TYPE (* IEC61131-3, Table 14#5 *)
  (* Standard: 1131-3 *)
  (* Version 0.0, 1/8/2024, Cheyan, Schneider Electric, Template *)
  PACKAGE Main;
  {SET_ATTRIBUTE(nxtDataType, QdpEwqSPB7qzzh+NTQEinmNZ98ZHkHWxvNuG/cIXeimh6FQ57YZhv3Rx0Sj2iL0jUJM+RBxfMAI=)}
  TimeAccuracy : (
    item1,
    item2,
    item3
  );
END_TYPE
